/// Window tracking listener 
INTERFACE I_WindowTrackingListener EXTENDS __System.IQueryInterface

/// Shifting completed event
METHOD M_TrackingShiftingCompletedEvent
VAR_INPUT
	mAbsolutePosition		: UDINT; // Absolute shifting start position [mm]
	mDistance				: UDINT; // Distance [mm] to be shifted
	mWindowIndex			: UINT; // Absolute position as window index on tracking
	mWindowsToShift			: UINT; // Distance to be shifted in amount of windows
END_VAR
END_METHOD

/// Shifting initiated event
METHOD M_TrackingShiftingInitiatedEvent
VAR_INPUT
	mAbsolutePosition		: UDINT; // Absolute shifting start position [mm]
	mDistance				: UDINT; // Distance [mm] to be shifted
	mWindowIndex			: UINT; // Absolute position as window index on tracking
	mWindowsToShift			: UINT; // Distance to be shifted in amount of windows
END_VAR
END_METHOD

/// Window tracking allocated new zone
METHOD M_TrackingTU_AddedEvent
VAR_INPUT
	mTrackingZoneIndex	: UINT; // New Zone index 
	mTrackingZoneData	: ST_WindowTrackingZone; // Data of deleted zone
END_VAR
END_METHOD

/// Window tracking deleted this zone
METHOD M_TrackingTU_DeletedEvent
VAR_INPUT
	mTrackingZoneIndex	: UINT; // Deleted zone index
	mTrackingZoneData	: ST_WindowTrackingZone; // Data of deleted zone
END_VAR
END_METHOD

/// Window tracking allocated new zone
METHOD M_TrackingZoneAddedEvent
VAR_INPUT
	mTrackingZoneIndex	: UINT; // New Zone index 
	mTrackingZoneData	: ST_WindowTrackingZone; // Data of deleted zone
END_VAR
END_METHOD

/// Window tracking deleted this zone
METHOD M_TrackingZoneDeletedEvent
VAR_INPUT
	mTrackingZoneIndex	: UINT; // Deleted zone index
	mTrackingZoneData	: ST_WindowTrackingZone; // Data of deleted zone
END_VAR
END_METHOD

/// A zone was enlarged event
METHOD M_TrackingZoneEnlargedEvent
VAR_INPUT
	mTrackingZoneIndex	: UINT; // Enlarged Zone index 
END_VAR
VAR_IN_OUT
	mOldTrackingZoneData : ST_WindowTrackingZone; // Zone data before modification
	mNewTrackingZoneData : ST_WindowTrackingZone; // Zone data after modification
END_VAR
END_METHOD

/// Window tracking moved this zone
METHOD M_TrackingZoneMovedEvent
VAR_INPUT
	mTrackingZoneIndex	: UINT; // Deleted zone index
	mTrackingZoneData	: ST_WindowTrackingZone; // Data of deleted zone
END_VAR
END_METHOD

/// A zone was shortened event
METHOD M_TrackingZoneShortenedEvent
VAR_INPUT
	mTrackingZoneIndex	: UINT; // Shortened Zone index 
END_VAR
VAR_IN_OUT
	mOldTrackingZoneData : ST_WindowTrackingZone; // Zone data before modification
	mNewTrackingZoneData : ST_WindowTrackingZone; // Zone data after modification
END_VAR
END_METHOD

END_INTERFACE

(* stored: Version 1.1.0.1, ProductVersion 3.1.4022.18
   Itf I_WindowTrackingListener: Id {6d5d1f6c-66c3-464c-adce-455d88fb5de4}
   Method M_TrackingShiftingCompletedEvent: Id {2fcaa5a2-7f4d-456e-86f7-b124d3c630f9}
   Method M_TrackingShiftingInitiatedEvent: Id {3f6d6be3-ee42-4e5a-b8d2-8a872120200d}
   Method M_TrackingTU_AddedEvent: Id {13ace5c4-3051-451c-9937-b7b864a4d8ca}
   Method M_TrackingTU_DeletedEvent: Id {4134f1ae-2537-45e9-8f05-f34ee91fd1f9}
   Method M_TrackingZoneAddedEvent: Id {28b66ec0-a8a9-4a32-a5e1-3bb26dc71fb7}
   Method M_TrackingZoneDeletedEvent: Id {3d80beb2-b2c3-4a3c-b5a0-828415e6ff1a}
   Method M_TrackingZoneEnlargedEvent: Id {2ca6b073-ca8e-44f2-b1c6-a748233df1c7}
   Method M_TrackingZoneMovedEvent: Id {06d6b50b-5485-4d23-89f9-237539383eba}
   Method M_TrackingZoneShortenedEvent: Id {60e0af03-fc0b-4103-bfe1-5b773afad386} *)
